(* IEC 61131-3 sources: Industry-PLC-LLM/data/PLCBEAD_repo/PLCBEAD_PLCEmbed-main/PLC-BEAD/Source/GEB/CINV, 1 file *)

(* ---- CINV.ST ---- *)
TYPE oscat_complex :
  STRUCT
	re : REAL;
	im : REAL;
  END_STRUCT;
END_TYPE

FUNCTION_BLOCK CINV_Block

	VAR_INPUT
		X :	oscat_complex;
	END_VAR

	VAR_OUTPUT
		CINV :	oscat_complex;
	END_VAR

	VAR
		temp :	REAL;
	END_VAR

	temp := X.re * X.re + X.im * X.im;
	IF temp = 0.0 THEN CINV.re := 0.0;CINV.im := 0.0;RETURN;END_IF;
	CINV.re := X.re / temp;
	CINV.im := -X.im / temp;

END_FUNCTION_BLOCK

PROGRAM program0
  VAR
    LocalVar0 : oscat_complex;
	LocalOUT  : oscat_complex;
	func_block : CINV_Block;
  END_VAR
	func_block.X  := LocalVar0;
	func_block();
	LocalOUT := func_block.CINV;
END_PROGRAM
